{region '#Template'}
	{attribute 'Version' := '6.0.0.0'}
	{attribute 'Tags' := '"LCID": "1031", "Text": "RA, Room, Sample"'}
	{attribute 'Tags' := '"LCID": "1033", "Text": "RA, Room, Sample"'}
	{attribute 'Using' := '"Type": "Template", "URI": "Site"'}
	{attribute 'Using' := '"Type": "Template", "URI": "BA2_Param"'}
	{attribute 'Using' := '"Type": "Template", "URI": "ST_BA_Facade"'}
	{attribute 'Using' := '"Type": "Template", "URI": "ST_BA_Lighting"'}
	{attribute 'Description' := '"LCID": "1031", "Text": "Beispiel Template Raum"'}
	{attribute 'Description' := '"LCID": "1033", "Text": "Sample-template room"'}
{endregion}
FUNCTION_BLOCK FB_BA_RoomSample1 EXTENDS FB_BA_View
VAR_INPUT
	stFacade					: ST_BA_Facade;			// sunblind-data from the next higher level
	stAreaLighting				: ST_BA_Lighting;		// lighting-data from the next higher level
END_VAR
		
VAR_INPUT CONSTANT PERSISTENT					
	{attribute 'parameterUnit':= 'KELVIN'}	                    
	fRmTAdjMin					: REAL;
	{attribute 'parameterUnit':= 'KELVIN'}	                    
	fRmTAdjMax					: REAL;
	{attribute 'parameterUnit':= 'KELVIN'}	                    
	fLgtT						: REAL;
	{attribute 'parameterUnit':= 's'}	                    
	nPollingIntervalFast		: UDINT;
	{attribute 'parameterUnit':= 's'}	                    
	nPollingIntervalNormal		: UDINT;
END_VAR	

VAR_INPUT CONSTANT
	BrtnsPrcSns					: FB_BA_BrightnessPresenceDALI;
	                    		
	Ctrl						: FB_BA_HeatCool_PID;
	VlvHtg						: FB_BA_ActuatorAnalog;
 	VlvCol						: FB_BA_ActuatorAnalog;
	                    		
	WdwCon1						: FB_BA_SensorBinary;
	WdwCon2						: FB_BA_SensorBinary;
	DewPointSensor				: FB_BA_SensorBinary;	
	RmTSen						: FB_BA_SensorAnalog;
	RmTAdj						: FB_BA_SensorAnalog;
	SunBldZone					: FB_BA_SunblindZone;
	SunBld1						: FB_BA_SunBld;		
	SunBld2						: FB_BA_SunBld;				
	LightZoneConstant			: FB_BA_LightGroupConstant;
	Light1						: FB_BA_LightAnalog;
	Light2						: FB_BA_LightAnalog;
END_VAR                 		
VAR                     		
	bSunbldSwiUp				: BOOL;
	bSunbldSwiDwn				: BOOL;	
	bLightSwi					: BOOL;	
	RmTAvg						: FB_BA_EnAvrg02;
	bInitializeSensor			: BOOL;	
END_VAR
VAR // added by the converter: edge detectors and wires of the graphical bodies
    _s1, _s2 : ST_BA_Analog;
END_VAR

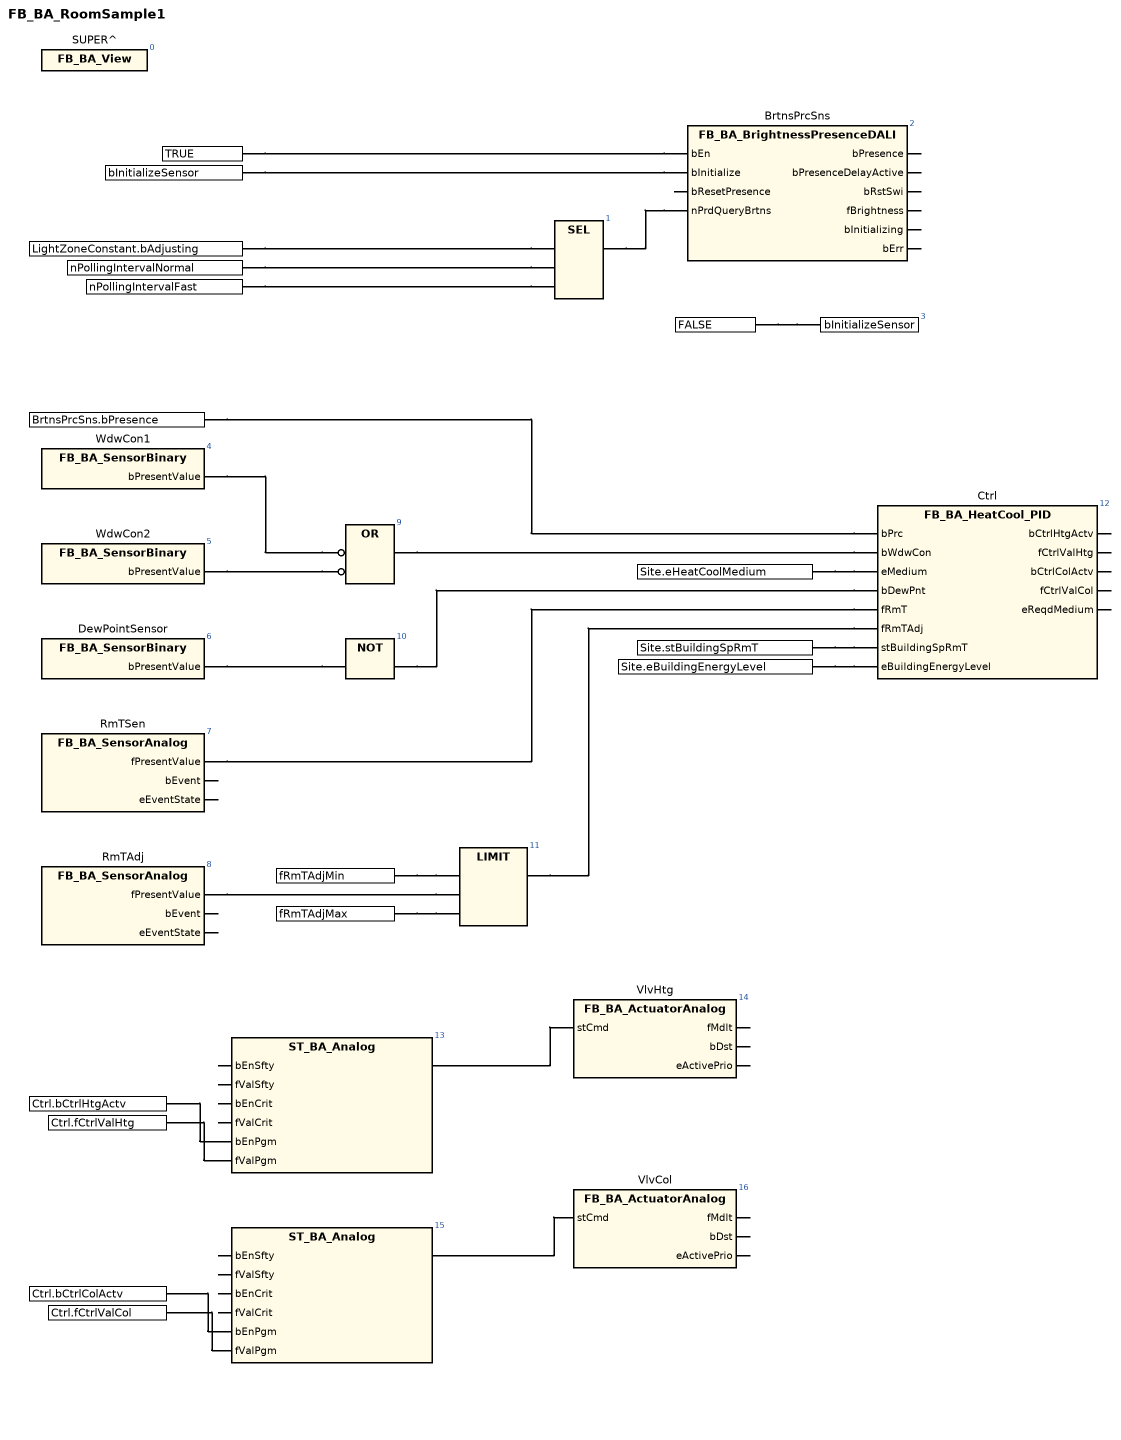
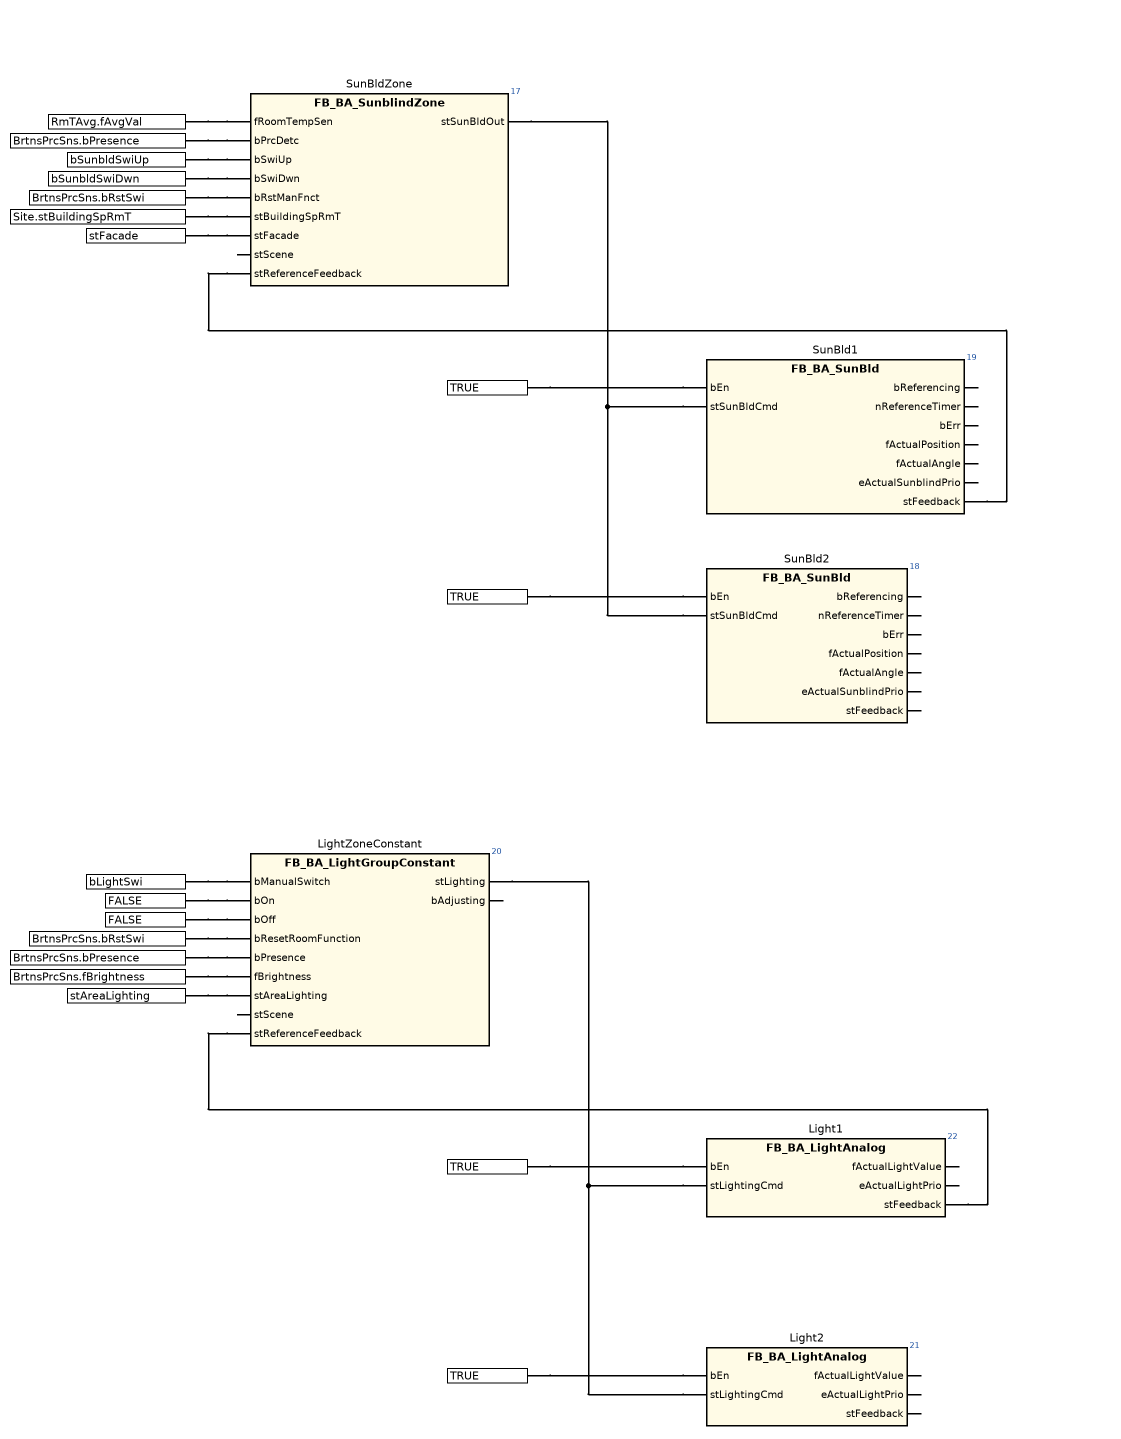
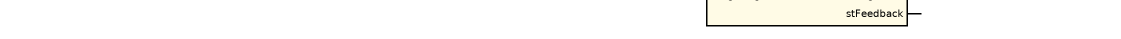
SUPER^(); // FB_BA_View
BrtnsPrcSns(
    bEn := TRUE,
    bInitialize := bInitializeSensor,
    nPrdQueryBrtns := SEL(LightZoneConstant.bAdjusting, nPollingIntervalNormal, nPollingIntervalFast)); // FB_BA_BrightnessPresenceDALI
bInitializeSensor := FALSE;
WdwCon1(); // FB_BA_SensorBinary
WdwCon2(); // FB_BA_SensorBinary
DewPointSensor(); // FB_BA_SensorBinary
RmTSen(); // FB_BA_SensorAnalog
RmTAdj(); // FB_BA_SensorAnalog
Ctrl(
    bPrc := BrtnsPrcSns.bPresence,
    bWdwCon := NOT WdwCon1.bPresentValue OR NOT WdwCon2.bPresentValue,
    eMedium := Site.eHeatCoolMedium,
    bDewPnt := NOT DewPointSensor.bPresentValue,
    fRmT := RmTSen.fPresentValue,
    fRmTAdj := LIMIT(fRmTAdjMin, RmTAdj.fPresentValue, fRmTAdjMax),
    stBuildingSpRmT := Site.stBuildingSpRmT,
    eBuildingEnergyLevel := Site.eBuildingEnergyLevel); // FB_BA_HeatCool_PID
// compose _s1 : ST_BA_Analog
_s1.bEnPgm := Ctrl.bCtrlHtgActv;
_s1.fValPgm := Ctrl.fCtrlValHtg;
VlvHtg(stCmd := _s1); // FB_BA_ActuatorAnalog
// compose _s2 : ST_BA_Analog
_s2.bEnPgm := Ctrl.bCtrlColActv;
_s2.fValPgm := Ctrl.fCtrlValCol;
VlvCol(stCmd := _s2); // FB_BA_ActuatorAnalog
SunBldZone(
    fRoomTempSen := RmTAvg.fAvgVal,
    bPrcDetc := BrtnsPrcSns.bPresence,
    bSwiUp := bSunbldSwiUp,
    bSwiDwn := bSunbldSwiDwn,
    bRstManFnct := BrtnsPrcSns.bRstSwi,
    stBuildingSpRmT := Site.stBuildingSpRmT,
    stFacade := stFacade,
    stReferenceFeedback := SunBld1.stFeedback); // FB_BA_SunblindZone
SunBld2(bEn := TRUE, stSunBldCmd := SunBldZone.stSunBldOut); // FB_BA_SunBld
SunBld1(bEn := TRUE, stSunBldCmd := SunBldZone.stSunBldOut); // FB_BA_SunBld
LightZoneConstant(
    bManualSwitch := bLightSwi,
    bOn := FALSE,
    bOff := FALSE,
    bResetRoomFunction := BrtnsPrcSns.bRstSwi,
    bPresence := BrtnsPrcSns.bPresence,
    fBrightness := BrtnsPrcSns.fBrightness,
    stAreaLighting := stAreaLighting,
    stReferenceFeedback := Light1.stFeedback); // FB_BA_LightGroupConstant
Light2(bEn := TRUE, stLightingCmd := LightZoneConstant.stLighting); // FB_BA_LightAnalog
Light1(bEn := TRUE, stLightingCmd := LightZoneConstant.stLighting); // FB_BA_LightAnalog

METHOD FB_init : BOOL
VAR_INPUT
	bInitRetains : BOOL; // if TRUE, the retain variables are initialized (warm start / cold start)
	bInCopyCode : BOOL;  // if TRUE, the instance afterwards gets moved into the copy code (online change)
END_VAR
BrtnsPrcSns.iParent							:= THIS^;
BrtnsPrcSns.iLabel							:= LblCtl_BrightnessPresenceSensor; 			
BrtnsPrcSns.eDPADMode						:= E_BA_DPADMode.eInclude;	
BrtnsPrcSns.nAdr							:= 11;
BrtnsPrcSns.nInstancePresence				:= 1;	
BrtnsPrcSns.nInstanceBrightness				:= 0;
BrtnsPrcSns.nResBrtns						:= 10;
BrtnsPrcSns.ipDALICommunication				:= DALICommunication.fbKL6821Communication;

nPollingIntervalFast						:= 1;			// fast interval polling the light-value e.g. in case of active light-adapting
nPollingIntervalNormal						:= 15;			// slow interval polling the light-value

WdwCon1.iParent								:= THIS^;
WdwCon1.iLabel								:= LblAgg_WindowContact; 			
WdwCon1.eDPADMode							:= E_BA_DPADMode.eInclude;		
WdwCon1.Input.iLabel						:= LblFun_Status; 	
WdwCon1.Input.ePolarity						:= E_BA_Polarity.eReverse;
WdwCon1.Input.sActiveText 					:= txtEvent_Closed;
WdwCon1.Input.sInactiveText 				:= txtEvent_Opened;
WdwCon1.Input.nEventClassID					:= EC_ID.NC50;
WdwCon1.Input.aEventTransitionText[1]		:= txtEvent_Disturb;
WdwCon1.Input.aEventTransitionText[2]		:= txtEvent_None;
WdwCon1.Input.aEventTransitionText[3]		:= txtEvent_Normal;
WdwCon1.Input.bEventDetectionEnable			:= FALSE;
                                    		
WdwCon2.iParent								:= THIS^;
WdwCon2.iLabel								:= LblAgg_WindowContact; 			
WdwCon2.eDPADMode							:= E_BA_DPADMode.eInclude;		
WdwCon2.Input.iLabel						:= LblFun_Status; 	
WdwCon2.Input.ePolarity						:= E_BA_Polarity.eReverse;
WdwCon2.Input.sActiveText 					:= txtEvent_Closed;
WdwCon2.Input.sInactiveText 				:= txtEvent_Opened;
WdwCon2.Input.nEventClassID					:= EC_ID.NC50;
WdwCon2.Input.aEventTransitionText[1]		:= txtEvent_Disturb;
WdwCon2.Input.aEventTransitionText[2]		:= txtEvent_None;
WdwCon2.Input.aEventTransitionText[3]		:= txtEvent_Normal;
WdwCon2.Input.bEventDetectionEnable			:= FALSE;

DewPointSensor.iParent						:= THIS^;
DewPointSensor.iLabel						:= LblAgg_MonitorDewPoint; 			
DewPointSensor.eDPADMode					:= E_BA_DPADMode.eInclude;		
DewPointSensor.Input.iLabel					:= LblFun_Status; 	
DewPointSensor.Input.ePolarity				:= E_BA_Polarity.eReverse;	
DewPointSensor.Input.sActiveText 			:= txtEvent_Normal;
DewPointSensor.Input.sInactiveText 			:= txtEvent_Triggered;
DewPointSensor.Input.nEventClassID			:= EC_ID.NC40;
DewPointSensor.Input.aEventTransitionText[1]:= txtEvent_Triggered;
DewPointSensor.Input.aEventTransitionText[2]:= txtEvent_None;
DewPointSensor.Input.aEventTransitionText[3]:= txtEvent_Normal;
DewPointSensor.Input.bEventDetectionEnable	:= TRUE;

RmTSen.iParent								:= THIS^;
RmTSen.iLabel								:= LblAgg_TemperatureRoomAir; 			
RmTSen.eDPADMode							:= E_BA_DPADMode.eInclude;		
RmTSen.MV.eUnit 							:= E_BA_Unit.eTemperature_DegreesCelsius;
RmTSen.MV.nEventClassID						:= EC_ID.NC60;
RmTSen.MV.aEventTransitionText[1]			:= txtEvent_Disturb;
RmTSen.MV.aEventTransitionText[2]			:= txtEvent_None;
RmTSen.MV.aEventTransitionText[3]			:= txtEvent_Normal;
RmTSen.MV.eEnPlantLock						:= E_BA_LockPriority.eNoLock;
RmTSen.MV.fResolution 						:= 0.01;
RmTSen.MV.fScaleOffset 						:= 0; 
                     			        	
RmTAdj.iParent								:= THIS^;
RmTAdj.iLabel								:= LblAgg_RoomControlUnit; 	
RmTAdj.eDPADMode							:= E_BA_DPADMode.eInclude;		
RmTAdj.MV.eUnit 							:= E_BA_Unit.eTemperature_DegreesKelvin;
RmTAdj.MV.nEventClassID						:= EC_ID.NC60;
RmTAdj.MV.aEventTransitionText[1]			:= txtEvent_Disturb;
RmTAdj.MV.aEventTransitionText[2]			:= txtEvent_None;
RmTAdj.MV.aEventTransitionText[3]			:= txtEvent_Normal;
RmTAdj.MV.eEnPlantLock						:= E_BA_LockPriority.eNoLock;
RmTAdj.MV.fResolution 						:= 0.01;
RmTAdj.MV.fScaleOffset 						:= 0; 
        
fRmTAdjMin									:= -5;	// limits of room-temperature-adjustment           
fRmTAdjMax									:= 5;	// in order to prevent adjusting from 0 to 50 degrees, for example

Ctrl.iParent								:= THIS^;
Ctrl.iLabel									:= LblCtl_RoomTemperatureControl; 			 
Ctrl.eDPADMode								:= E_BA_DPADMode.eInclude;

VlvHtg.iParent								:= THIS^;
VlvHtg.iLabel								:= LblAgg_Valve; 	
VlvHtg.eDPADMode							:= E_BA_DPADMode.eInclude;
VlvHtg.Mdlt.eUnit 							:= E_BA_Unit.eOther_Percent;
VlvHtg.Mdlt.nEventClassID					:= EC_ID.NC60;
VlvHtg.Mdlt.aEventTransitionText[1]			:= txtEvent_Disturb;
VlvHtg.Mdlt.aEventTransitionText[2]			:= txtEvent_None;
VlvHtg.Mdlt.aEventTransitionText[3]			:= txtEvent_Normal;		
VlvHtg.Mdlt.fResolution 					:= 0.01;
VlvHtg.Mdlt.fScaleOffset 					:= 0; 		 
                            			    
VlvCol.iParent								:= THIS^;
VlvCol.iLabel								:= LblAgg_Valve; 	
VlvCol.eDPADMode							:= E_BA_DPADMode.eInclude;
VlvCol.Mdlt.eUnit 							:= E_BA_Unit.eOther_Percent;
VlvCol.Mdlt.nEventClassID					:= EC_ID.NC60;
VlvCol.Mdlt.aEventTransitionText[1]			:= txtEvent_Disturb;
VlvCol.Mdlt.aEventTransitionText[2]			:= txtEvent_None;
VlvCol.Mdlt.aEventTransitionText[3]			:= txtEvent_Normal;		
VlvCol.Mdlt.fResolution 					:= 0.01;
VlvCol.Mdlt.fScaleOffset 					:= 0; 



SunBldZone.iParent							:= THIS^;
SunBldZone.iLabel							:= LblCtl_SunblindZoneControl; 		

Sunbld1.iParent								:= THIS^;
Sunbld1.iLabel								:= LblCtl_SunblindActuator; 	
Sunbld1.sObjectName							:= '{Idx=01}';		 		 
Sunbld1.eDPADMode							:= E_BA_DPADMode.eInclude;

Sunbld2.iParent								:= THIS^;
Sunbld2.iLabel								:= LblCtl_SunblindActuator; 	
Sunbld2.sObjectName							:= '{Idx=02}';	 		 
Sunbld2.eDPADMode							:= E_BA_DPADMode.eInclude;



Light1.iParent								:= THIS^;
Light1.iLabel								:= LblCtl_LightActuator; 	
Light1.sObjectName							:= '{Idx=01}';		 
Light1.eDPADMode							:= E_BA_DPADMode.eInclude;

Light2.iParent								:= THIS^;
Light2.iLabel								:= LblCtl_LightActuator; 		
Light2.sObjectName							:= '{Idx=02}';	 
Light2.eDPADMode							:= E_BA_DPADMode.eInclude;

LightZoneConstant.iParent					:= THIS^;
LightZoneConstant.iLabel					:= LblCtl_LightZoneControl; 			 
LightZoneConstant.eDPADMode					:= E_BA_DPADMode.eInclude;

fLgtT										:= 3000;		// light-temperature [K]
END_METHOD

END_FUNCTION_BLOCK

(* stored: Version 1.1.0.1, ProductVersion 3.1.4024.13
   POU FB_BA_RoomSample1: Id {1e7b8644-8a3c-4605-8c9d-d7f0bbbd293f}, SpecialFunc None
   Method FB_init: Id {a4cd8cb6-cb78-40e0-88f8-74a5eb466d7b} *)
